FUNCTION F_RecJointData : ST_JointData									// Different for different structures
VAR_INPUT
	data: ARRAY [1..500] OF BYTE;
END_VAR
VAR
	nNumOfVar: UINT;
	nIndex: UINT;
	pAddrTo: POINTER TO ST_JointData;
	PAddrFrom: POINTER TO ARRAY [1..500] OF BYTE;
	nByteCount: UINT;
	
	n2Byte : UINT;
	n4Byte : UDINT;
	n8Byte : ULINT;
	adr2Byte: POINTER TO UINT;
	adr4Byte: POINTER TO UDINT;
	adr8Byte: POINTER TO ULINT;
	nCurrentVarLength: USINT;
END_VAR

nNumOfVar := SIZEOF(F_RecJointData.arrVarLength);						// Different for different structures
pAddrTo := ADR(F_RecJointData);											// Different for different structures
PAddrFrom := ADR(data);
nByteCount := 0;
adr2Byte := ADR(n2Byte);
adr4Byte := ADR(n4Byte);
adr8Byte := ADR(n8Byte);

FOR nIndex := 1 TO nNumOfVar DO
	nCurrentVarLength := F_RecJointData.arrVarLength[nIndex];			// Different for different structures
	
	(* Determine byte address to save item to *)
	nByteCount := nByteCount + nCurrentVarLength;
	IF nByteCount=8 THEN
		pAddrTo := pAddrTo;
		nByteCount := 0;
	ELSIF nByteCount>8 THEN
		pAddrTo := pAddrTo + 16 - nByteCount;
		nByteCount := 0;
	ELSE
		pAddrTo := pAddrTo;
	END_IF
	
	(* Convert Data based on size of item (in bytes) *)
	IF nCurrentVarLength=8 THEN
		MEMCPY(adr8Byte, pAddrFrom, 8);
		n8Byte := BE64_TO_HOSTEX(n8Byte);
		MEMCPY(pAddrTo, adr8Byte, 8);
	ELSIF nCurrentVarLength=4 THEN
		MEMCPY(adr4Byte, pAddrFrom, 8);
		n4Byte := BE32_TO_HOST(n4Byte);
		MEMCPY(pAddrTo, adr4Byte, 8);
	ELSIF nCurrentVarLength=2 THEN
		MEMCPY(adr2Byte, pAddrFrom, 8);
		n2Byte := BE16_TO_HOST(n2Byte);
		MEMCPY(pAddrTo, adr2Byte, 8);
	ELSE
		MEMCPY( pAddrTo, pAddrFrom, nCurrentVarLength);
	END_IF
	
	(* Increment addressed of interest *)
	pAddrFrom := PAddrFrom + nCurrentVarLength;
	pAddrTo := pAddrTo + nCurrentVarLength;
END_FOR

END_FUNCTION

(* stored: Version 1.1.0.1, ProductVersion 3.1.4020.12
   POU F_RecJointData: Id {36dcd17e-b4da-4855-8055-5a9bc102e5cb}, SpecialFunc None *)
